TYPE
    ST_MyComponent_Config_1 : STRUCT
        ExtendTime  : LREAL;
        RetractTime : LREAL;
    END_STRUCT
END_TYPE

(* stored: Version 1.1.0.1
   DUT ST_MyComponent_Config_1: Id {d89d8c7d-e826-4b04-8701-15331f22b4d9} *)
